(* IEC 61131-3 sources: Industry-PLC-LLM/data/PLCBEAD_repo/PLCBEAD_PLCEmbed-main/PLC-BEAD/Source/GEB/MAX_TIME, 1 file *)

(* ---- MAX_TIME.ST ---- *)
FUNCTION _MAX_TIME:TIME

	VAR_INPUT
		IN1 :	TIME;
		IN2 :	TIME;
	END_VAR

	_MAX_TIME := SEL_TIME(IN1 < IN2,IN1,IN2);

END_FUNCTION

PROGRAM program0
	VAR
		IN1 :	TIME;
		IN2 :	TIME;

		OUT : TIME;
	END_VAR

	OUT := _MAX_TIME(IN1, IN2);

END_PROGRAM
